FUNCTION_BLOCK CU00xManual EXTENDS TcoCore.TcoTask
VAR
END_VAR

IF(THIS^.Execute())THEN
	;
END_IF

PROPERTY Station : REFERENCE TO CU00x
GET
VAR
    _station : POINTER TO CU00x;
END_VAR
IF __QUERYPOINTER(Parent,_station) THEN // Check if _Parent is Station001
	Station REF= _station^;              // If the check is successful dereference a pointer. simlar to THIS^ or SUPER^
END_IF
END_GET
END_PROPERTY

END_FUNCTION_BLOCK

(* stored: Version 1.1.0.1, ProductVersion 3.1.4024.9
   POU CU00xManual: Id {4da1dfbc-4c0a-47a8-95b6-4f0ca8024493}, SpecialFunc None
   Property Station: Id {400a1f67-80cb-4f9f-a632-be597ac0ffc5}
   Get Get: Id {e3aceaef-61ff-438d-83cd-a8c6edd964ba} *)
